INTERFACE I_SynchronousRpcResponse EXTENDS I_Disposable

METHOD PUBLIC CompleteWithBase64
VAR_INPUT
	pBytes : POINTER TO BYTE;
	nBytes : DINT;
END_VAR
END_METHOD

METHOD PUBLIC CompleteWithBool
VAR_INPUT
	Value : BOOL;
END_VAR
END_METHOD

METHOD PUBLIC CompleteWithBytesAsHex
VAR_INPUT
	pBytes : POINTER TO BYTE;
	nBytes : DINT;
END_VAR
END_METHOD

METHOD PUBLIC CompleteWithDateTime
VAR_INPUT
	Value : DATE_AND_TIME;
END_VAR
END_METHOD

METHOD PUBLIC CompleteWithDcTime
VAR_INPUT
	Value : DCTIME;
END_VAR
END_METHOD

METHOD PUBLIC CompleteWithDint
VAR_INPUT
	Value : DINT;
END_VAR
END_METHOD

METHOD PUBLIC CompleteWithFileTime
VAR_INPUT
	Value : FILETIME;
END_VAR
END_METHOD

METHOD PUBLIC CompleteWithLint
VAR_INPUT
	Value : LINT;
END_VAR
END_METHOD

METHOD PUBLIC CompleteWithLreal
VAR_INPUT
	Value : LREAL;
END_VAR
END_METHOD

METHOD PUBLIC CompleteWithNull
VAR_INPUT
END_VAR
END_METHOD

METHOD PUBLIC CompleteWithObject
VAR_INPUT
	Object : I_Serializable;
END_VAR
END_METHOD

METHOD PUBLIC CompleteWithReal
VAR_INPUT
	Value : REAL;
END_VAR
END_METHOD

METHOD PUBLIC CompleteWithSerializer
VAR_INPUT
	Serializer : I_Serializer;
END_VAR
END_METHOD

METHOD PUBLIC CompleteWithString
VAR_INPUT
	Value : T_MAXSTRING;
END_VAR
END_METHOD

METHOD PUBLIC CompleteWithUdint
VAR_INPUT
	Value : UDINT;
END_VAR
END_METHOD

METHOD PUBLIC CompleteWithUlint
VAR_INPUT
	Value : ULINT;
END_VAR
END_METHOD

METHOD PUBLIC GetSerializer : I_Serializer
VAR_INPUT
END_VAR
END_METHOD

METHOD PUBLIC RejectWithError
VAR_INPUT
	ErrorCode : T_MAXSTRING;
	Message : T_MAXSTRING;
END_VAR
END_METHOD

METHOD PUBLIC TryMakeAsynchronous : BOOL
VAR_INPUT
	Destination : REFERENCE TO I_AsynchronousRpcResponse;
END_VAR
END_METHOD

END_INTERFACE

(* stored: Version 1.1.0.1, ProductVersion 3.1.4026.13
   Itf I_SynchronousRpcResponse: Id {f4b0555e-5337-4cdc-be55-8b26f12c4521}
   Method CompleteWithBase64: Id {e2b6083b-2e5f-45aa-8c2c-8748b4544107}
   Method CompleteWithBool: Id {cfd2c6aa-f1da-436c-bf59-6beda70e7a2e}
   Method CompleteWithBytesAsHex: Id {c7976d47-f065-46d3-b74c-3ceae82fdf02}
   Method CompleteWithDateTime: Id {824b7474-b7f0-4587-919b-d0fe6612f160}
   Method CompleteWithDcTime: Id {77e2c395-3f02-4d20-94c8-79a9115f3c0f}
   Method CompleteWithDint: Id {556fff2e-96e6-4647-b555-967f1648df59}
   Method CompleteWithFileTime: Id {09dcb5d1-ec49-4568-bea8-f33e0c0ab29f}
   Method CompleteWithLint: Id {85cc9cfa-d31d-45f3-a904-b78d018b7f66}
   Method CompleteWithLreal: Id {5aab574d-1acf-4b19-9677-95af87a2c7e6}
   Method CompleteWithNull: Id {a99067be-444a-4c0b-be3b-5f1d57be4bf6}
   Method CompleteWithObject: Id {50ee507a-f405-431e-bca3-afe5fe56ef04}
   Method CompleteWithReal: Id {5860ea5f-0dc6-42db-8881-d5fd6173000b}
   Method CompleteWithSerializer: Id {f9c508d4-79b6-4773-99a6-d56a7441b19c}
   Method CompleteWithString: Id {493e0770-0c2d-4885-8d96-1810bc14b946}
   Method CompleteWithUdint: Id {371838ee-997e-4ca2-924b-7c6bcea82dcf}
   Method CompleteWithUlint: Id {7f33f1fe-7124-45c5-be13-e09f8c3a6cf9}
   Method GetSerializer: Id {fc5a7a74-aa05-426a-8299-b3c7f7ef1e04}
   Method RejectWithError: Id {aab767f6-f9bb-41de-910d-0b93655ca1d1}
   Method TryMakeAsynchronous: Id {a8486bd6-d182-4261-a066-aa4950a3667d} *)
